{attribute addProperty BoxType "EJ2521-0224-0016"}
{attribute addProperty Id "Target_counter_valueAT %Q*UINT162"}
{attribute addProperty CRC "3356238523"}
{attribute addProperty SizeInBites "16"}
{attribute addProperty SizeInBytes "2"}
TYPE PTO_Target_compact_C80C22BB :
STRUCT
	{attribute addProperty Name "Target_counter_value"}
	Target_counter_value AT %Q* : UINT;
END_STRUCT
END_TYPE

(* stored: Version 1.2.0.0, ProductVersion 3.1.4024.9
   DUT PTO_Target_compact_C80C22BB: Id {50216fce-a555-48b5-a968-d796f7620449} *)
